{attribute 'GeneratedUsingTerminal: KL1644-0050'}
{attribute addProperty BoxType "KL1644-0050"}
{attribute addProperty Id "SwitchAT %I*BOOL0OutputAT %Q*BOOL0"}
{attribute addProperty CRC "1802648086"}
{attribute addProperty Size "0"}
TYPE Channel_6B723A16 :
STRUCT
	{attribute addProperty Name "Switch"}
	Switch AT %I* : BOOL;
	{attribute addProperty Name "Output"}
	Output AT %Q* : BOOL;
END_STRUCT
END_TYPE

(* stored: Version 1.2.0.0, ProductVersion 3.1.4024.9
   DUT Channel_6B723A16: Id {3edfaede-661d-4034-80ca-ecbc44b1f814} *)
